// TIA Portal V21 export
VAR_GLOBAL   // PLC tag table "K_Macchinario"
END_VAR
VAR_GLOBAL CONSTANT   // user constants
   K_CodiceMacchinario_SterilizzatoreTubo : Int := 010102;   // 01 Processo e trattamento - 01 Termico - 02 SterilizzatoreTubo
   K_CodiceMacchinario_Spiedinatrice : Int := 010301;   // 01 Processo e trattamento - 03 Meccanico - 01 Spiedinatrice
END_VAR
